TYPE ST_ClampStationOutCmd :
STRUCT
    CycleCompleted : BOOL;
END_STRUCT
END_TYPE

(* stored: Version 1.1.0.1, ProductVersion 3.1.4024.12
   DUT ST_ClampStationOutCmd: Id {d536924a-f414-4817-83f5-11445c39e593} *)
